TYPE sc_db_Set_Work_Order_WaitLoading_Pos :
STRUCT
	uuid : STRING(36);
	Pos : LREAL;
END_STRUCT
END_TYPE

(* stored: Version 1.1.0.1, ProductVersion 3.1.4026.13
   DUT sc_db_Set_Work_Order_WaitLoading_Pos: Id {15775541-c828-4fa7-b973-0ac129d9baaa} *)
